Staubli VAL3: FC_InitMotion.pgx

program FC_InitMotion()
begin
  //this function is goiong to begin synchronous motion
  $movejSyncBegin(mNomSpeed)
end
